// TwinCAT 3 PLC project SPS
// ProgramVersion: 3.1.4024.0
// libraries:
//   Tc2_MC2, * (Beckhoff Automation GmbH)
//   Tc2_Standard, * (Beckhoff Automation GmbH)
//   Tc2_System, * (Beckhoff Automation GmbH)
//   Tc3_IotBase, * (Beckhoff Automation GmbH)
//   Tc3_Module, * (Beckhoff Automation GmbH)
// project tree:
//   DUTs/ State.TcDUT, State_Dispenser.TcDUT, State_Foerderband.TcDUT, State_Motorsteuerung.TcDUT, State_Motor_Manipulator.TcDUT, State_Vereinzelung.TcDUT
//   GVLs/ IFC_HW.TcGVL (not stored)
//   / PlcTask.TcTTO
//   POUs/FBs/ FB_Blink.TcPOU, FB_Conveyor.TcPOU, FB_Dispenser.TcPOU, FB_Foerderband.TcPOU, FB_Manipulator.TcPOU, FB_MQTT.TcPOU, FB_StatusLight.TcPOU, FB_Vereinzelung.TcPOU
//   POUs/ MAIN.TcPOU
// real-time tasks:
//   TASK PlcTask: cycle T#10ms, priority 20, ADS port 350
// motion (NC):
//   TASK NC-Task 1 SAF: cycle T#2ms, priority 4, ADS port 501
//   TASK NC-Task 1 SVB: cycle T#10ms, priority 8, ADS port 511
//   AXIS BandMotor (id 1)
//     Dynamic: AccelerationMaximum=700, DecelerationMaximum=700, Acceleration=500, Deceleration=500
//     Velo: Maximum=50
//     OtherSettings: AllowMotionCmdToSlave=true
//     encoder EncType=1
//     drive DrvType=5
//       Analog: VeloReferenz=57, TorqueSetpointScale=10, ScaleFactorActTorque=0.1
//       TimeComp: TaskDelayCycles=1
//     controller CtrType=1
//       CtrPara: PriorControlFactor=1
//         Observer: BandWidth=20
//   AXIS Extruder1 (id 2)
//     OtherSettings: AllowMotionCmdToSlave=true
//     encoder EncType=1
//     drive DrvType=5
//       Analog: TorqueSetpointScale=10, ScaleFactorActTorque=0.1
//       TimeComp: TaskDelayCycles=1
//     controller CtrType=1
//       CtrPara: PriorControlFactor=1
//         Observer: BandWidth=20
//   AXIS Extruder2 (id 3)
//     OtherSettings: AllowMotionCmdToSlave=true
//     encoder EncType=1
//     drive DrvType=5
//       Analog: TorqueSetpointScale=10, ScaleFactorActTorque=0.1
//       TimeComp: TaskDelayCycles=1
//     controller CtrType=1
//       CtrPara: PriorControlFactor=1
//         Observer: BandWidth=20
//   AXIS Extruder3 (id 4)
//     OtherSettings: AllowMotionCmdToSlave=true
//     encoder EncType=1
//     drive DrvType=5
//       Analog: TorqueSetpointScale=10, ScaleFactorActTorque=0.1
//       TimeComp: TaskDelayCycles=1
//     controller CtrType=1
//       CtrPara: PriorControlFactor=1
//         Observer: BandWidth=20
//   AXIS ManX (id 5)
//     OtherSettings: AllowMotionCmdToSlave=true
//     encoder EncType=1
//     drive DrvType=5
//       Analog: TorqueSetpointScale=10, ScaleFactorActTorque=0.1
//       TimeComp: TaskDelayCycles=1
//     controller CtrType=1
//       CtrPara: PriorControlFactor=1
//         Observer: BandWidth=20
//   AXIS ManY (id 6)
//     OtherSettings: AllowMotionCmdToSlave=true
//     encoder EncType=1
//     drive DrvType=5
//       Analog: TorqueSetpointScale=10, ScaleFactorActTorque=0.1
//       TimeComp: TaskDelayCycles=1
//     controller CtrType=1
//       CtrPara: PriorControlFactor=1
//         Observer: BandWidth=20
//   AXIS ManZ (id 7)
//     OtherSettings: AllowMotionCmdToSlave=true
//     encoder EncType=1
//     drive DrvType=5
//       Analog: TorqueSetpointScale=10, ScaleFactorActTorque=0.1
//       TimeComp: TaskDelayCycles=1
//     controller CtrType=1
//       CtrPara: PriorControlFactor=1
//         Observer: BandWidth=20
//   AXIS Greifer (id 8)
//     OtherSettings: AllowMotionCmdToSlave=true
//     encoder EncType=1
//     drive DrvType=5
//       Analog: TorqueSetpointScale=10, ScaleFactorActTorque=0.1
//       TimeComp: TaskDelayCycles=1
//     controller CtrType=1
//       CtrPara: PriorControlFactor=1
//         Observer: BandWidth=20
// variable links:
//   SPS/SPS Instance <-> NC-Task 1 SAF/Axes/BandMotor
//     PlcTask Inputs/IFC_HW.ax_BandMotor.NcToPlc <-> Outputs/ToPlc
//     PlcTask Outputs/IFC_HW.ax_BandMotor.PlcToNc <-> Inputs/FromPlc
//   SPS/SPS Instance <-> NC-Task 1 SAF/Axes/Extruder1
//     PlcTask Inputs/IFC_HW.ax_Extruder1.NcToPlc <-> Outputs/ToPlc
//     PlcTask Outputs/IFC_HW.ax_Extruder1.PlcToNc <-> Inputs/FromPlc
//   SPS/SPS Instance <-> NC-Task 1 SAF/Axes/Extruder2
//     PlcTask Inputs/IFC_HW.ax_Extruder2.NcToPlc <-> Outputs/ToPlc
//     PlcTask Outputs/IFC_HW.ax_Extruder2.PlcToNc <-> Inputs/FromPlc
//   SPS/SPS Instance <-> NC-Task 1 SAF/Axes/Extruder3
//     PlcTask Inputs/IFC_HW.ax_Extruder3.NcToPlc <-> Outputs/ToPlc
//     PlcTask Outputs/IFC_HW.ax_Extruder3.PlcToNc <-> Inputs/FromPlc
//   SPS/SPS Instance <-> NC-Task 1 SAF/Axes/Greifer
//     PlcTask Inputs/IFC_HW.ax_ManG.NcToPlc <-> Outputs/ToPlc
//     PlcTask Outputs/IFC_HW.ax_ManG.PlcToNc <-> Inputs/FromPlc
//   SPS/SPS Instance <-> NC-Task 1 SAF/Axes/ManX
//     PlcTask Inputs/IFC_HW.ax_ManX.NcToPlc <-> Outputs/ToPlc
//     PlcTask Outputs/IFC_HW.ax_ManX.PlcToNc <-> Inputs/FromPlc
//   SPS/SPS Instance <-> NC-Task 1 SAF/Axes/ManY
//     PlcTask Inputs/IFC_HW.ax_ManY.NcToPlc <-> Outputs/ToPlc
//     PlcTask Outputs/IFC_HW.ax_ManY.PlcToNc <-> Inputs/FromPlc
//   SPS/SPS Instance <-> NC-Task 1 SAF/Axes/ManZ
//     PlcTask Inputs/IFC_HW.ax_ManZ.NcToPlc <-> Outputs/ToPlc
//     PlcTask Outputs/IFC_HW.ax_ManZ.PlcToNc <-> Inputs/FromPlc

CONFIGURATION SPS
    RESOURCE PLC ON TwinCAT3
        TASK PlcTask(INTERVAL := T#10ms, PRIORITY := 20);
        PROGRAM MAIN WITH PlcTask : MAIN;
    END_RESOURCE
END_CONFIGURATION

// ---- DUTs/State.TcDUT
{attribute 'qualified_only'}
{attribute 'strict'}
TYPE State :
(
	Off,
	Init,
	Ready,
	Production,
	Done,
	Error,
	Stop,
	Setup
);
END_TYPE

// ---- DUTs/State_Dispenser.TcDUT
{attribute 'qualified_only'}
{attribute 'strict'}
TYPE State_Dispenser :
(
	Off,
	Reset, 
	Reset_done,
	Power, 
	Ready, 
	Dispensing,
	Done,
	Wait
);
END_TYPE

// ---- DUTs/State_Foerderband.TcDUT
{attribute 'qualified_only'}
{attribute 'strict'}
TYPE State_Foerderband :
(
	Off,
	Power_up,
	Ready,
	Move_to_next,
	Wait,
	Done,
	Error,
	wait_for_next
);
END_TYPE

// ---- DUTs/State_Motorsteuerung.TcDUT
{attribute 'qualified_only'}
{attribute 'strict'}
TYPE State_Motorsteuerung :
(
	Off,
	Reset,
	Power,
	Ready,
	Moving
);
END_TYPE

// ---- DUTs/State_Motor_Manipulator.TcDUT
{attribute 'qualified_only'}
{attribute 'strict'}
TYPE State_Motor_Manipulator :
(
	OFF,
	INIT,
	RESET,
	READY,
	REF,
	PRODUCTION
);
END_TYPE

// ---- DUTs/State_Vereinzelung.TcDUT
{attribute 'qualified_only'}
{attribute 'strict'}
TYPE State_Vereinzelung :
(
	Off,
	Check,
	Init,
	Init_wait,
	Bereit,	
	Auswerfen,
	Auswerfen_wait,
	Fertig
);
END_TYPE

// ---- POUs/MAIN.TcPOU
PROGRAM MAIN
VAR
	
    fbStatusLight : FB_StatusLight;
    fbVereinzelung : FB_Vereinzelung;
    fbFoerderband : FB_Foerderband;
	fbDispenser1 : FB_Dispenser;
	fbDispenser2 : FB_Dispenser;
	fbDispenser3 : FB_Dispenser;
	fbManipulator : FB_Manipulator;
	fbIot : FB_MQTT;

    bEnable : BOOL := FALSE;
    bExecute : BOOL := FALSE;
    nState_main : INT := 0;
    timer : TON;
	timer2 : TON;
	timer3 : TON;
	timer4 : TON;
	timer5 : TON;
	timer6 : TON;
	timer7 : ton;
	
	nTargetPosX : INT := 100; // Beispielwert
    nTargetPosY : INT := 200; // Beispielwert
    nTargetPosZ : INT := 300; // Beispielwert
	
END_VAR

// Zuweisung der globalen Variablen
bEnable := IFC_HW.bEnable;
bExecute := IFC_HW.bExecute;

// Initialisierung der Funktionsbausteine mit den globalen Variablen
fbStatusLight(eStatus := fbManipulator.eStatus, bRed => bAmpelRot, bYellow => bAmpelGelb, bGreen => bAmpelGrun);

fbIot();

fbVereinzelung(
    bSensor_1 := bEinzelSens1, 
    bSensor_2 := bEinzelSens2,
    bAkt1_1 => bR2AKT1,
    bAkt1_2 => bR1AKT1,
    bAkt2_1 => bR2AKT2,
    bAkt2_2 => bR1AKT2
);

fbFoerderband(
	bSensor1:= IFC_HW.bBandSens1, 
	bSensor2:= IFC_HW.bBandSens2, 
	bSensor3:= IFC_HW.bBandSens3, 
	bSensor4:= IFC_HW.bBandSens4, 
	ax :=  IFC_HW.ax_BandMotor, 
	bStopper1=> IFC_HW.bBandHub1, 
	bStopper2=> IFC_HW.bBandHub2, 
	bStopper3=> IFC_HW.bBandHub3
	);

fbDispenser1( 
    ax := IFC_HW.ax_Extruder1
);

fbDispenser2( 
    ax := IFC_HW.ax_Extruder2
);

fbDispenser3( 
    ax := IFC_HW.ax_Extruder3
);

fbManipulator(
    nTargetPositionX := nTargetPosX,
    nTargetPositionY := nTargetPosY,
    nTargetPositionZ := nTargetPosZ,
    axX := IFC_HW.ax_ManX,
    axY := IFC_HW.ax_ManY,
    axZ := IFC_HW.ax_ManZ
);

fbDispenser1.nDispenceGram := 5;
fbDispenser2.nDispenceGram := 2;
fbDispenser3.nDispenceGram := 7;

IF NOT bEnable THEN
    nState_main := 0;
END_IF

CASE nState_main OF
    0:  // Off
        fbVereinzelung.bEnable := FALSE;
        fbFoerderband.bEnable := FALSE;
		fbDispenser1.bEnable := FALSE;
		fbDispenser2.bEnable := FALSE;
		fbDispenser3.bEnable := FALSE;
		fbManipulator.bEnable := FALSE;

        IF bEnable THEN 
            nState_main := 1;
        END_IF

    1:  // Turn on
        fbVereinzelung.bEnable := TRUE;
  		fbFoerderband.bEnable := TRUE;
		fbDispenser1.bEnable := TRUE;
		fbDispenser2.bEnable := TRUE;
		fbDispenser3.bEnable := TRUE;
		fbManipulator.bEnable := TRUE;
		fbManipulator.bHome := TRUE;

        IF fbVereinzelung.eStatus = State.Ready  AND fbFoerderband.eStatus = State.Ready AND fbDispenser1.eStatus = State.Ready AND fbDispenser2.eStatus = State.Ready AND fbDispenser3.eStatus = State.Ready THEN
            nState_main := nState_main + 1;
        END_IF

    2:  // Vereinzeln
        IF bExecute THEN
            fbVereinzelung.bExecute := TRUE;
            IF fbVereinzelung.eStatus = State.Production THEN
                fbVereinzelung.bExecute := FALSE;
				nState_main := nState_main + 1;
            END_IF
        END_IF

	3:	// Fahre zu pos. 1
		fbFoerderband.bExecute := TRUE;		
		IF fbFoerderband.eStatus = State.Done THEN
			fbFoerderband.bExecute := FALSE;
			timer(in := TRUE, pt := T#2S);
			IF timer.q THEN
				timer.IN := FALSE;
				nState_main := nState_main + 1;
			END_IF 
		END_IF
		
	4: // Starte Dispenser 1
		fbDispenser1.bExecute := TRUE;
		IF fbDispenser1.bDone THEN
			fbDispenser1.bExecute := FALSE;
			nState_main := nState_main + 1;
		END_IF
		
	5:	// warte
		timer2(in := TRUE, pt := T#2S);
		IF timer2.Q THEN
			timer2.IN := FALSE;
			nState_main := nState_main + 1;
		END_IF
	
	6: 	// fahre zu pos. 2
		fbFoerderband.bExecute := TRUE;
		timer3(in := TRUE, pt := T#2S);
		IF timer3.Q THEN
			timer3.IN := FALSE;
			fbFoerderband.bExecute := FALSE;
			nState_main := nState_main + 1;
		END_IF
		
		
	7: // warte
		IF fbFoerderband.eStatus = State.Done THEN
			timer(in := TRUE, pt := T#4S);
			IF timer.Q THEN
				nState_main := nState_main + 1;
			END_IF
		END_IF
		
	8:	// starte dispenser 2
		fbDispenser2.bExecute := TRUE;
		IF fbDispenser2.eStatus = State.Done THEN
			fbDispenser2.bExecute := FALSE;
			nState_main := nState_main + 1;
		END_IF
		
	9:	// warte
		timer(in := TRUE, pt := T#2S);
		IF timer.Q THEN
			timer.IN := FALSE;
			nState_main := nState_main + 1;
		END_IF
		
	10:	// fahre zu pos 3
		fbFoerderband.bExecute := TRUE;
		timer5(in := TRUE, pt := T#2S);
		IF timer5.Q THEN
			timer5.IN := FALSE;
			fbFoerderband.bExecute := FALSE;
			nState_main := nState_main + 1;
		END_IF
	
	11: //komme an pos 3 an
		IF fbFoerderband.eStatus = State.Done THEN
			nState_main := nState_main + 1;
		END_IF
		
	12: // starte dispenser 3
		fbDispenser3.bExecute := TRUE;
		IF fbDispenser3.eStatus = State.Done THEN
			fbDispenser3.bExecute := FALSE;
			nState_main := nState_main + 1;
		END_IF
		
	13:	// warte
		fbFoerderband.bExecute := TRUE;
		timer6(in := TRUE, pt := T#2S);
		IF timer6.Q THEN
			fbFoerderband.bExecute := FALSE;
			nState_main := nState_main + 1;
		END_IF
		
	14: // komme an pos 4 an
		IF fbFoerderband.bEnd_Foerderband THEN
			nState_main := nState_main + 1;
		END_IF
		
	15:	//fahre auf position
		fbManipulator.nTargetPositionX := 29;
		fbManipulator.nTargetPositionY := 145.5;
		fbManipulator.nTargetPositionZ := 45;
		fbManipulator.bMoveToPosition := TRUE;
		
		IF fbManipulator.bDone THEN
			nState_main := nState_main +1;
			fbManipulator.bMoveToPosition := FALSE;
		END_IF
		
		
	16: // warte
		timer7(in := TRUE, pt := T#2S);
		IF timer7.Q THEN
			timer7.IN := FALSE;
			nState_main := nState_main +1;
		END_IF
		
	17: // fahre zu flasche runter
		
		//fbManipulator.nTargetPositionX := 29;
		//fbManipulator.nTargetPositionY := 145.5;
		//fbManipulator.nTargetPositionZ := 130;
		//fbManipulator.bMoveToPosition := TRUE;
		
		
		
		
		
		
		
		
		
		
END_CASE

END_PROGRAM

// ---- POUs/FBs/FB_StatusLight.TcPOU
FUNCTION_BLOCK FB_StatusLight
VAR_INPUT

	eStatus : State;	

END_VAR
VAR_OUTPUT
	
	bGreen : BOOL;
	bYellow : BOOL;
	bRed : BOOL;
	
END_VAR
VAR
	
	fbBlink : FB_Blink;

END_VAR

fbBlink(bStart := TRUE);

CASE eStatus OF
	State.Done :
	bRed := FALSE;
	bGreen := TRUE;
	bYellow := TRUE;
	
	State.Error:
	bRed := fbBlink.bBlink;
	bGreen := FALSE;
	bYellow := FALSE;
	
	State.Init:
	bGreen := fbBlink.bBlink;
	bRed := FALSE;
	bYellow := FALSE;
	
	State.Off :
	bGreen := FALSE;
	bRed := TRUE;
	bYellow := FALSE;
	
	State.Stop :
	bGreen := FALSE;
	bRed := fbBlink.bBlink;
	bYellow := fbBlink.bBlink;
	
	State.Production :
	bGreen := TRUE;
	bRed := FALSE;
	bYellow := FALSE;
	
	
	State.Ready :
	bGreen := fbBlink.bBlink;
	bRed := FALSE;
	bYellow := TRUE;
END_CASE

END_FUNCTION_BLOCK

// ---- POUs/FBs/FB_Blink.TcPOU
FUNCTION_BLOCK FB_Blink
VAR_INPUT
	
	bStart : BOOL := FALSE;
	
END_VAR
VAR_OUTPUT
	
	bBlink : BOOL := FALSE;
	
END_VAR
VAR
	
	fbPulse : TP;

END_VAR

fbPulse(IN := bStart AND NOT fbPulse.Q, PT := T#1S);

IF (fbPulse.ET <= fbPulse.PT/2) THEN
	bBlink := FALSE;
ELSE
	bBlink := TRUE;
END_IF

END_FUNCTION_BLOCK

// ---- POUs/FBs/FB_Vereinzelung.TcPOU
FUNCTION_BLOCK FB_Vereinzelung
VAR_INPUT
	
	bEnable : BOOL;
	bExecute : BOOL;
	bSensor_1 : BOOL;
	bSensor_2 : BOOL;
	bSensor_3 : bool;
	
END_VAR

VAR_OUTPUT
	
	bAkt1_1 : BOOL;		// Akteur oben schließen
	bAkt1_2 : BOOL;		// Akteur oben öffnen
	
	bAkt2_1 : BOOL;		// Akteur unten schließen
	bAkt2_2 : BOOL;		// Akteur unten öffnen
	
	eStatus : State := State.Off;	// State-Machine Anzeige
	
END_VAR

VAR
	
	timer_schleusse_1 : TON;
	timer_schleusse_2 : TON;
	eState_vereinzelung : State_Vereinzelung := State_Vereinzelung.Off;
	
END_VAR

timer_schleusse_1(PT := T#2S); // Timer mit 2s
timer_schleusse_2(PT := T#5S); // Timer mit 5s

CASE eState_vereinzelung OF
	State_Vereinzelung.Off:
	
	eStatus := State.Off;
	
	// beide schleußen zu
	bAkt1_1 :=	TRUE;
	bAkt1_2 :=	FALSE;
	bAkt2_1 :=	TRUE;
	bAkt2_2 :=	FALSE;
	
	IF bEnable THEN
		eState_vereinzelung := State_Vereinzelung.Check;
		
	END_IF
	
	// überprüfe status von Vereinzelung
	State_Vereinzelung.Check:
	
	eStatus := State.Off;	// immer noch aus
	
	bAkt1_1 :=	TRUE;
	bAkt1_2 :=	FALSE;
	bAkt2_1 :=	TRUE;
	bAkt2_2 :=	FALSE;
	
	IF bSensor_2 THEN
		eState_vereinzelung := State_Vereinzelung.Init;
	END_IF
	
	// Initialisieren State, öffne obere Schleuße
	State_Vereinzelung.Init:
	
	eStatus := State.Init;
	
	// öffne obere schleuße
	bAkt1_1 :=	FALSE;
	bAkt1_2 :=	TRUE;
	bAkt2_1 :=	TRUE;
	bAkt2_2 :=	FALSE;
	
	IF bSensor_1 THEN
		eState_vereinzelung := State_Vereinzelung.Init_wait;
	END_IF
	
	// warte bis die obere schleuße zu ist (timer)
	State_Vereinzelung.Init_wait:
	
	bAkt1_1 :=	TRUE;
	bAkt1_2 :=	FALSE;
	bAkt2_1 :=	TRUE;
	bAkt2_2 :=	FALSE;
	
	timer_schleusse_1.IN := TRUE;
	
	IF timer_schleusse_1.Q THEN
		timer_schleusse_1.IN := FALSE;
		eState_vereinzelung := State_Vereinzelung.Bereit;
	END_IF
	
	// Bereit zum flasche auszuwerfen
	State_Vereinzelung.Bereit:
	
	eStatus := State.Ready;
	
	bAkt1_1 :=	TRUE;
	bAkt1_2 :=	FALSE;
	bAkt2_1 :=	TRUE;
	bAkt2_2 :=	FALSE;
	
	IF bExecute and not bSensor_3 THEN
		eState_vereinzelung := State_Vereinzelung.Auswerfen;
	END_IF
	
	// Flasche auswerfen
	State_Vereinzelung.Auswerfen:
	
	eStatus := State.Production;
	
	bAkt1_1 :=	TRUE;
	bAkt1_2 :=	FALSE;
	bAkt2_1 :=	FALSE;
	bAkt2_2 :=	TRUE;
	
	IF NOT bSensor_1 THEN
		eState_vereinzelung := State_Vereinzelung.Auswerfen_wait;
	END_IF
	
	// warten nach auswerfen dass Flasche wirklich weg ist
	State_Vereinzelung.Auswerfen_wait:
	
	timer_schleusse_2.IN := TRUE;
	
	IF timer_schleusse_2.Q THEN
		timer_schleusse_2.IN := FALSE;
		eState_vereinzelung := State_Vereinzelung.Fertig;
	END_IF
	
	// Flasche ist weg, Schleuße wieder schließen
	State_Vereinzelung.Fertig:
	
	eStatus := State.Done;
	
	// schleuße 2 wieder zu fahren
	bAkt1_1 :=	TRUE;
	bAkt1_2 :=	FALSE;
	bAkt2_1 :=	TRUE;
	bAkt2_2 :=	FALSE;
	
	timer_schleusse_1.IN := TRUE;
	
	IF timer_schleusse_1.Q AND NOT bExecute THEN
		timer_schleusse_1.IN := FALSE;
		eState_vereinzelung := State_Vereinzelung.Check;
	END_IF
	
END_CASE

END_FUNCTION_BLOCK

// ---- POUs/FBs/FB_Foerderband.TcPOU
FUNCTION_BLOCK FB_Foerderband
VAR_INPUT
	
	bEnable : BOOL; //enables FB
	bExecute : BOOL; // transport the flask one position further
	
	bSensor1 : BOOL;
	bSensor2 : BOOL;
	bSensor3 : BOOL;
	bSensor4 : BOOL;
	
END_VAR
VAR_OUTPUT

	bEnd_Foerderband : BOOL := FALSE;	

	eStatus : State := State.Off;
	
	bStopper1: BOOL;
	bStopper2: BOOL;
	bStopper3: BOOL;
	
END_VAR
VAR_IN_OUT
	
	ax : AXIS_REF;
	
END_VAR
VAR
	
	//Conveyer FB
	fbConveyor : FB_Conveyor;
	
	//internal state
	eState_foerderband : State_Foerderband := State_Foerderband.Off;
	
	//counter of current position
	nCurrentPosition_1 : INT := 0;
	nCurrentPosition_2 : INT := 0;
	
	//timer
	timer:TON;
	
END_VAR

fbConveyor(
	ax := ax);
	
CASE eState_foerderband OF
	State_Foerderband.Off:
		eStatus := State.Off;
		
		bStopper1 := FALSE;
		bStopper2 := FALSE;
		bStopper3 := FALSE;
		
		fbConveyor.bEnable := FALSE;
	
		IF bEnable THEN
		fbConveyor.bEnable := TRUE;
		eState_foerderband := State_Foerderband.Power_up;
		END_IF
	
	State_Foerderband.Power_up:
		IF fbConveyor.eStatus = State.Ready THEN
			eState_foerderband := State_Foerderband.Ready;
		END_IF
		
	State_Foerderband.Ready:
		bStopper1 := FALSE;
		bStopper2 := FALSE;
		bStopper3 := FALSE;
		eStatus := State.Ready;
		IF bExecute THEN
			eState_foerderband := State_Foerderband.Move_to_next;
		END_IF
		
	State_Foerderband.Move_to_next:
		eStatus := State.Production;
		fbConveyor.bStop := FALSE;
		fbConveyor.bExecute := TRUE;
		CASE nCurrentPosition_1 OF
			0: 
			IF bSensor1 THEN
				nCurrentPosition_2 :=0;
				eState_foerderband := State_Foerderband.Wait;
			END_IF
			1: 
				bStopper1 := TRUE;
				IF bSensor2  AND NOT bSensor1 THEN
					nCurrentPosition_2 :=1;
					eState_foerderband := State_Foerderband.Wait;
				END_IF
			2: 
				bStopper1 := FALSE;
				bStopper2 := TRUE;
				IF bSensor3 THEN
					nCurrentPosition_2 :=2;
					eState_foerderband := State_Foerderband.Wait;
				END_IF
			3: 
				bStopper2 := FALSE;
				bStopper3 := TRUE;
				IF bSensor4 THEN
					bEnd_Foerderband := TRUE;
					nCurrentPosition_2 :=3;
					eState_foerderband := State_Foerderband.Wait;
				END_IF
		END_CASE
		
	State_Foerderband.Wait:
		timer(IN:=TRUE, PT:=T#1S);
		IF timer.Q THEN
			timer(IN:=FALSE);
			eState_foerderband := State_Foerderband.Done;
			bStopper1 := FALSE;
			bStopper2 := FALSE;
			bStopper3 := FALSE;
		END_IF
		
	State_Foerderband.Done:
		eStatus := State.Done;
		CASE nCurrentPosition_2 OF
			0: 
				fbConveyor.bExecute := FALSE;
				fbConveyor.bStop := TRUE;
				nCurrentPosition_1 :=1;
			1: 
				fbConveyor.bExecute := FALSE;
				fbConveyor.bStop := TRUE;
				nCurrentPosition_1 :=2;
			2: 
				fbConveyor.bExecute := FALSE;
				fbConveyor.bStop := TRUE;
				nCurrentPosition_1 :=3;
					
			3: 
				fbConveyor.bExecute := FALSE;
				fbConveyor.bStop := TRUE;
				nCurrentPosition_1 :=0;
				bEnd_Foerderband := FALSE;
		END_CASE
		
		eState_foerderband := State_Foerderband.wait_for_next;
		
		
	State_Foerderband.wait_for_next:
		IF bExecute THEN // warten solange von aussen bexecute geschaltet wird. wird getan sobald disp1,2,3 fertig ist	
			eState_foerderband := State_Foerderband.Move_to_next;
		END_IF
		

	
END_CASE

END_FUNCTION_BLOCK

// ---- POUs/FBs/FB_Conveyor.TcPOU
FUNCTION_BLOCK FB_Conveyor
VAR_INPUT
    bEnable  : BOOL;
    bExecute : BOOL;
	bStop : BOOL;
END_VAR

VAR_IN_OUT
    ax : AXIS_REF;  // Achsen Referenz
END_VAR

VAR_OUTPUT
    eStatus : State;
END_VAR

VAR
    fbPower : MC_Power;
    fbMoveVelocity : MC_MoveVelocity;
    fbHalt : MC_Halt;
    bAxPower : BOOL;
    bAxMove : BOOL;
    bHalt : BOOL;

    eState_conveyor : INT := 0;
END_VAR

// Achse updaten
ax.ReadStatus();

// Achsenfreigabe (Power) aufrufen
fbPower(Axis := ax, Enable := bAxPower, Enable_Positive := TRUE, Enable_Negative := TRUE);

// Bewegungsbefehl aufrufen
fbMoveVelocity(Axis := ax, Execute := bAxMove, Velocity := 30, Direction := Mc_Positive_Direction);

// Haltbefehl aufrufen
fbHalt(Axis := ax, Execute := bHalt);

IF NOT bEnable THEN
    eState_conveyor := 0;
    eStatus := State.Off;
    bAxPower := FALSE;
    bAxMove := FALSE;
    bHalt := TRUE;
ELSE
    CASE eState_conveyor OF
        0: // Off
            eStatus := State.Off;
            bAxPower := FALSE;
            bAxMove := FALSE;
            bHalt := TRUE;
            IF bEnable THEN
                eState_conveyor := 1;
            END_IF

        1: // Powering up
            eStatus := State.Init;
            bAxPower := TRUE;
            IF fbPower.Status THEN
                eState_conveyor := 2;
            END_IF

        2: // Ready
            eStatus := State.Ready;
			bHalt := TRUE;
            bAxMove := FALSE;
            IF bExecute THEN
				bHalt := false;
                eState_conveyor := 3;
            END_IF

        3: // Production
            eStatus := State.Production;
            bAxMove := TRUE;
            IF bStop THEN   
				bHalt := TRUE;
				bAxMove := FALSE;             
				eState_conveyor := 2;
			END_IF
    END_CASE
END_IF

END_FUNCTION_BLOCK

// ---- POUs/FBs/FB_Dispenser.TcPOU
FUNCTION_BLOCK FB_Dispenser
VAR_INPUT
    bEnable      : BOOL;
    bExecute     : BOOL;
    nDispenceGram: REAL;
END_VAR

VAR_IN_OUT
    ax : AXIS_REF;  // Achsen Referenz
END_VAR

VAR_OUTPUT
    eStatus : State;
    bDone   : BOOL;
END_VAR

VAR
    fbPower        : MC_Power;
    fbMoveDistance : MC_MoveRelative;
    fbHalt         : MC_Halt;
    bAxPower       : BOOL;
    bAxMove        : BOOL;
    bHalt          : BOOL;
    nDistance      : REAL;
	nVelocity 	   : REAL := 50;
    eState_dispenser : INT := 0;
    doneTimer      : TON;
END_VAR

// Berechne die Bewegungsdistanz
nDistance := (nDispenceGram * 50);

// Achse updaten
ax.ReadStatus();

// Achsenfreigabe (Power) aufrufen
fbPower(Axis := ax, Enable := bAxPower, Enable_Positive := TRUE, Enable_Negative := TRUE);

// Bewegungsbefehl aufrufen
fbMoveDistance(Axis := ax, Execute := bAxMove, Distance := nDistance, Velocity := nVelocity);

// Haltbefehl aufrufen
fbHalt(Axis := ax, Execute := bHalt);

IF NOT bEnable THEN
    eState_dispenser := 0;
    eStatus := State.Off;
    bAxPower := FALSE;
    bAxMove := FALSE;
    bHalt := TRUE;
    bDone := FALSE;
ELSE
    CASE eState_dispenser OF
        0: // Off
            eStatus := State.Off;
            bAxPower := FALSE;
            bAxMove := FALSE;
            bHalt := TRUE;
            bDone := FALSE;
            IF bEnable THEN
                eState_dispenser := 1;
            END_IF

        1: // Powering up
            eStatus := State.Init;
            bAxPower := TRUE;
            IF fbPower.Status THEN
                eState_dispenser := 2;
            END_IF

        2: // Ready
            eStatus := State.Ready;
            bAxMove := FALSE;
            bHalt := FALSE;
            bDone := FALSE;
            IF bExecute THEN
                eState_dispenser := 3;
            END_IF

        3: // Production
            eStatus := State.Production;
            bAxMove := TRUE;
            bHalt := FALSE;
            
            IF fbMoveDistance.Done THEN
                bAxMove := FALSE;
                bDone := TRUE;
				eStatus := State.Done;
                eState_dispenser := 4;
            END_IF

        4: // Done, waiting to reset
			doneTimer(IN := TRUE, PT := T#2S);
            IF doneTimer.Q THEN
                doneTimer.IN := FALSE;
                bDone := FALSE;
                eState_dispenser := 2; // Zurück zu Ready
            END_IF
    END_CASE
END_IF

END_FUNCTION_BLOCK

// ---- POUs/FBs/FB_Manipulator.TcPOU
FUNCTION_BLOCK FB_Manipulator

VAR_INPUT
    bEnable : BOOL;
    bMoveToPosition : BOOL;
    bHome : BOOL; 
    nTargetPositionX : REAL;
    nTargetPositionY : REAL;
    nTargetPositionZ : REAL;
END_VAR

VAR_OUTPUT
    eStatus : State;
    bDone : BOOL;
    bHomed : BOOL; 
END_VAR

VAR_IN_OUT
    axX : AXIS_REF;
    axY : AXIS_REF;
    axZ : AXIS_REF;
END_VAR

VAR
    fbPowerX : MC_Power;
    fbPowerY : MC_Power;
    fbPowerZ : MC_Power;
    fbMoveX : MC_MoveAbsolute;
    fbMoveY : MC_MoveAbsolute;
    fbMoveZ : MC_MoveAbsolute;
    fbHomeX : MC_Home;
    fbHomeY : MC_Home;
    fbHomeZ : MC_Home;
    mcResetX : MC_Reset;
    mcResetY : MC_Reset;
    mcResetZ : MC_Reset;
    bPowerOn : BOOL;
    eState_Manipulator : INT := 0;
    eState_Homing : INT := 0;
END_VAR

axX.ReadStatus();
axY.ReadStatus();
axZ.ReadStatus();

fbMoveX(
	Axis := axX, 
	Velocity := 40.0,
	Acceleration := 5.0,
	Deceleration := 5.0,	
	);
	
fbMoveY(
	Axis := axY, 
	Velocity := 40.0,
	Acceleration := 5.0,
	Deceleration := 5.0,	
	);
	
fbMoveZ(
	Axis := axZ, 
	Velocity := 40.0,
	Acceleration := 5.0,
	Deceleration := 5.0,	
	);


CASE eState_Manipulator OF
    0: // Off
        eStatus := State.Off;
        bPowerOn := FALSE;
        bDone := FALSE;
        bHomed := FALSE;

        IF bEnable THEN
            eState_Manipulator := 1;
        END_IF

    1: // Powering up
        bPowerOn := TRUE;
        fbPowerX(Axis := axX, Enable := bPowerOn, Enable_Positive := TRUE, Enable_Negative := TRUE);
        fbPowerY(Axis := axY, Enable := bPowerOn, Enable_Positive := TRUE, Enable_Negative := TRUE);
        fbPowerZ(Axis := axZ, Enable := bPowerOn, Enable_Positive := TRUE, Enable_Negative := TRUE);

        axX.ReadStatus();
        axY.ReadStatus();
        axZ.ReadStatus();

        IF fbPowerX.Status AND fbPowerY.Status AND fbPowerZ.Status THEN
            bPowerOn := FALSE;
            eState_Manipulator := 10;
        END_IF

    10: // Reset Axes X, Y, Z
        mcResetX(Axis := axX, Execute := TRUE);
        mcResetY(Axis := axY, Execute := TRUE);
        mcResetZ(Axis := axZ, Execute := TRUE);

        IF mcResetX.Done AND mcResetY.Done AND mcResetZ.Done THEN
            mcResetX.Execute := FALSE;
            mcResetY.Execute := FALSE;
            mcResetZ.Execute := FALSE;
            eState_Manipulator := 20;
        END_IF

    20: // Re-enable Axes X, Y, Z
        fbPowerX(Axis := axX, Enable := TRUE, Enable_Positive := TRUE, Enable_Negative := TRUE);
        fbPowerY(Axis := axY, Enable := TRUE, Enable_Positive := TRUE, Enable_Negative := TRUE);
        fbPowerZ(Axis := axZ, Enable := TRUE, Enable_Positive := TRUE, Enable_Negative := TRUE);

        IF fbPowerX.Status AND fbPowerY.Status AND fbPowerZ.Status THEN
            eState_Manipulator := 40;
        END_IF

    40: // Homing
        eStatus := State.Init;
        CASE eState_Homing OF
            0: // H0me X
                fbHomeX(Axis := axX, Execute := TRUE, HomingMode := MC_DefaultHoming, Position := 29, bCalibrationCam := bManEndXmin);
                IF fbHomeX.Done THEN
                    fbHomeX.Execute := FALSE;
                    eState_Homing := 1;
                END_IF

            1: // H0me Y
                fbHomeY(Axis := axY, Execute := TRUE, HomingMode := MC_DefaultHoming, Position := 145.5, bCalibrationCam := bManEndYmin);
                IF fbHomeY.Done THEN
                    fbHomeY.Execute := FALSE;
                    eState_Homing := 2;
                END_IF

            2: // Home Z
                fbHomeZ(Axis := axZ, Execute := TRUE, HomingMode := MC_DefaultHoming, Position := 45, bCalibrationCam := bManEndZmin);
                IF fbHomeZ.Done THEN
                    fbHomeZ.Execute := FALSE;
                    bHomed := TRUE;
                    eState_Manipulator := 3;
                END_IF
        END_CASE

    3: // Ready
        eStatus := State.Ready;
        IF bMoveToPosition THEN
            fbMoveX(Axis := axX, Position := nTargetPositionX, Execute := TRUE);
            fbMoveY(Axis := axY, Position := nTargetPositionY, Execute := TRUE);
            fbMoveZ(Axis := axZ, Position := nTargetPositionZ, Execute := TRUE);
            eState_Manipulator := 4;
        END_IF

    4: // Moving to position
        eStatus := State.Production;
        IF fbMoveX.Done AND fbMoveY.Done AND fbMoveZ.Done THEN
            eState_Manipulator := 5;
        END_IF

    5: // Done
        eStatus := State.Done;
        bDone := TRUE;
        IF NOT bMoveToPosition THEN
            eState_Manipulator := 3;
        END_IF

END_CASE

END_FUNCTION_BLOCK

// ---- POUs/FBs/FB_MQTT.TcPOU
FUNCTION_BLOCK FB_MQTT
VAR_INPUT
	sNamen_gr : STRING;
END_VAR
VAR_OUTPUT
END_VAR
VAR
	s_topic_prefix : STRING := 'aut/Ibk MQTTea Party/';
	
	fbMqttClient: FB_IotMqttClient; // MQTT client.
    TopicToPublish : STRING(255) := 'TwinCat/Temperatures'; // Mqtt topic on which we will broadcast the acual temperatures
    MessageToPublish : STRING(255); //String to send.
    fbSendMessageIntervalTimer : TON := (PT:=T#10S); //Interval timer for broadcasting.

    //ai_RoomTemperature AT %I* : INT; //Actual room temperature, linked to thermocouple
    ai_RoomTemperature : INT := 1; //Actual room temperature, linked to thermocouple
END_VAR

IF _TaskInfo[GETCURTASKINDEXEX()].FirstCycle THEN
    fbMqttClient.sHostName := '158.180.44.197';
    fbMqttClient.nHostPort := 1883;
    fbMqttClient.sTopicPrefix := s_topic_prefix;
    fbMqttClient.sClientId := 'Publishing PLC';
    fbMqttClient.sUserName      := 'bobm';
    fbMqttClient.sUserPassword  := 'letmein'; 
	
	fbMqttClient.Execute(bConnect := TRUE);
	
	
	
	MessageToPublish := 'Kloepfer, Pohle, Wild';
    fbMqttClient.Publish(sTopic:= 'names',
		pPayload:= ADR(MessageToPublish),
		nPayloadSize:= LEN(MessageToPublish)+1,
		eQoS:= TcIotMqttQos.AtMostOnceDelivery,
		bRetain:= TRUE,
		bQueue:= FALSE);
			
	MessageToPublish := 'IBK MQTTea Party';
    fbMqttClient.Publish(sTopic:= '$$groupsname',
		pPayload:= ADR(MessageToPublish),
		nPayloadSize:= LEN(MessageToPublish)+1,
		eQoS:= TcIotMqttQos.AtMostOnceDelivery,
		bRetain:= TRUE,
		bQueue:= FALSE);
		
	MessageToPublish := 'meter';
	fbMqttClient.Publish(sTopic:= 'Fuellstand/$$unit',
		pPayload:= ADR(MessageToPublish),
		nPayloadSize:= LEN(MessageToPublish)+1,
		eQoS:= TcIotMqttQos.AtMostOnceDelivery,
		bRetain:= TRUE,
		bQueue:= FALSE);
			
END_IF

fbMqttClient.Execute(bConnect := TRUE);

IF fbMqttClient.bConnected THEN
    fbSendMessageIntervalTimer(IN:=TRUE);
    IF fbSendMessageIntervalTimer.Q THEN
        fbSendMessageIntervalTimer(IN:=FALSE);
        MessageToPublish := REAL_TO_STRING(ai_RoomTemperature / 10.0);

        fbMqttClient.Publish(sTopic:= 'Fuellstand',
            pPayload:= ADR(MessageToPublish),
            nPayloadSize:= LEN(MessageToPublish)+1,
            eQoS:= TcIotMqttQos.AtMostOnceDelivery,
            bRetain:= TRUE,
            bQueue:= FALSE);
			
			
    END_IF
END_IF

END_FUNCTION_BLOCK
